DATA_BLOCK "Total_DB"
{ S7_Optimized_Access := 'FALSE' }
VERSION : 0.1
NON_RETAIN
   STRUCT
      Total_Reset_HMI : Bool;
      Restart_PLC : Bool;
   END_STRUCT;


BEGIN
   Total_Reset_HMI := FALSE;
   Restart_PLC := FALSE;

END_DATA_BLOCK

